// TIA Portal V18 export
VAR_GLOBAL   // PLC tag table "24_ESP-EG2"
   "iESP-EG2" AT %I13.1 : Bool;
   "oESP-EG2" AT %Q12.4 : Bool;
END_VAR
